PROGRAM P_Machine 

VAR	
	// MachineConfig
	stCurMachineConfig				: ST_MachineConfig;
	fOverride						: LREAL;
	bCheckPosBeforeRun				: BOOL;
	
	/// Sequences	
	seqOpMode						: FB_Sequence;
	
	bMaintMat						: BOOL;
	bMaintTool						: BOOL;
	stPunchJob						: ST_PunchJob;
		
	/// Components	
	fbComponents					: FB_CompositionBase;

	// PunchParameters
	bMatLoaded						: BOOL;
	bContinuous						: BOOL;
	nCurRun							: UINT;
	nCurPunch						: UDINT;
	nCurMat							: UINT;	
	nCurMoveOverride				: REAL;
	
	fThresholdX						: LREAL;
	fThresholdY						: LREAL;
	
	stCoordinate					: ST_Coordinate;
	stNextCoordinate				: ST_Coordinate;
	nMaxPunches						: UDINT;
	
	fMaxDisplacementX				: LREAL;
	fMaxDisplacementY				: LREAL;
	
	bInitialized					: BOOL;
	eJobState						: E_JobState;
	
	rtSafety						: R_TRIG;
	
	bSafeDrive						: BOOL;
	
	
END_VAR

// Init
Init();

bSafeDrive := fbSafety.SafetyOk AND fbSafetyLock.SafetyOk;

rtSafety(CLK:= NOT fbSafety.SafetyOk);

// SAFETY
IF rtSafety.Q THEN
	bInitialized := FALSE;
	seqOpMode.Start(E_OperationMode.eOperationMode_Halt);
	fbEventLog.WriteInfo(E_Event.eEvent_none, 'NOT HALT');
	
	IF eJobState = E_JobState.eJobState_running THEN
		eJobState := E_JobState.eJobState_stopped;
	END_IF
	
END_IF

// Run Components
fbEventLog.Run();
fbComponents.Run();

// Run Sequencer
seqOpMode.Enable := TRUE;
seqOpMode.Base(TRUE,FALSE);
CASE seqOpMode.SequenceId OF	
	E_OperationMode.eOperationMode_Maintenance:		_Maintenance();
	E_OperationMode.eOperationMode_Start:			_Start();
	E_OperationMode.eOperationMode_Stop:			_Stop();
	E_OperationMode.eOperationMode_Reset:			_Reset();
	E_OperationMode.eOperationMode_Halt:			_Halt();
END_CASE

METHOD _Halt : BOOL
VAR_INPUT
END_VAR
seqOpMode.Name := 'Halt';

CASE seqOpMode.Step OF
	
0	 :	seqOpMode.StepDefinition('Move to Zero Position', T#0S);
		fbPunchEngine.Halt();
		fbMatAndToolHandling.Halt();
		seqOpMode.NextStepDelay(T#1S, 10);	
		
10	 :	//fbSafetyLock.Unlock();
		seqOpMode.Finish();
		
END_CASE
END_METHOD

METHOD _Maintenance : BOOL
VAR_INPUT
END_VAR
seqOpMode.Name := 'Maintenance';

CASE seqOpMode.Step OF
	

0	 :	seqOpMode.StepDefinition('Move PunchEngine to Maint Position', T#0S);	
		fbPunchEngine.MoveTDC();			
		fbPunchEngine.OutletBeltseq(FALSE, 0);
		seqOpMode.NextStep(10);
	
10	 :	IF fbPunchEngine.TDC THEN
			seqOpMode.NextStep(20);		
		END_IF
		
20	 :	seqOpMode.StepDefinition('Move XY to Maint Position', T#0S);	
		fbMatAndToolHandling.MaintPos(NOT bMaintMat, NOT bMaintTool);	
		seqOpMode.NextStep(30);			
	
30	 :	IF fbMatAndToolHandling.TargetReached THEN 	
			seqOpMode.Finish();		
			//fbSafetyLock.Unlock();
		END_IF

			
END_CASE
END_METHOD

METHOD _Reset : BOOL
VAR_INPUT
END_VAR
CASE seqOpMode.Step OF

	0:	seqOpMode.StepDefinition('reset, init reset WF', T#0S);
		
		fbSafetyLock.Lock();
		bInitialized := FALSE;
		fbComponents.ResetComponents(FALSE, FALSE, 0, 0);
		
		fbEventLog.Mute := TRUE;
		fbEventLog.Reset();	
		
		seqOpMode.NextStepDelay(T#200MS, 10);	// skip safety

	10:	seqOpMode.StepDefinition('Reset: wait for request', T#0S);
		fbSafety.Reset();
		seqOpMode.NextStep(20);
		
	20:	seqOpMode.StepDefinition('Reset safety', T#0S);
		seqOpMode.NextStepTransition(30, fbSafety.State = E_ComponentState.eComponentState_running);
	
	30:	seqOpMode.StepDefinition('Reset all components', T#0S);
		fbComponents.ResetComponents(FALSE, FALSE, eComponentType_none, eComponentType_Safety);
		seqOpMode.NextStep(40);
		
	40:	seqOpMode.StepDefinition('wait for components ready...', T#0S);
		seqOpMode.NextStepTransitionDelay(fbComponents.CompostitionState = E_ComponentState.eComponentState_running, T#5S,  50);
		
	50:	seqOpMode.StepDefinition('Move to Zero Position', T#0S);
		fbPunchEngine.MoveTDC();
		fbPunchEngine.OutletBeltseq(FALSE, 0);
		seqOpMode.NextStep(60);	
		
	60:	IF fbPunchEngine.TDC THEN
			seqOpMode.NextStep(70);	
		END_IF
			
	70:	seqOpMode.StepDefinition('Finish', T#0S);
		fbEventLog.Mute := FALSE;
		fbEventLog.Reset();
		bInitialized := TRUE;
		seqOpMode.Finish();
		
END_CASE
END_METHOD

METHOD _Start : BOOL
VAR
	fTime				: LREAL;
	stTmpPosition		: ST_Coordinate;
END_VAR
seqOpMode.Name := 'Start';

CASE seqOpMode.Step OF
	
/// MAT LOOP

0	 :	seqOpMode.StepDefinition('Check Mat', T#0S);
		
		fbSafetyLock.Lock();
		IF NOT bInitialized THEN			// AUTO INIT
			seqOpMode.NextSequenceId := eOperationMode_Start;
			seqOpMode.Start(E_operationMode.eOperationMode_Reset);
			RETURN;
		END_IF
		
		IF NOT fbMatAndToolHandling.Ready OR NOT fbPunchEngine.Ready THEN
			RETURN;
		END_IF

		IF nCurMat > MATS_COUNT THEN
			fbPunchEngine.MoveTDC();
			fbMatAndToolHandling.MoveRelX(stCurMachineConfig.fMoveOutside ,stCurMachineConfig.fVelocityX, stCurMachineConfig.fAccelerationX);
			fbEventLog.WriteInfo(E_Event.eEvent_none, 'no further Mat Found');
			seqOpMode.NextStep(5);		
			RETURN;
		END_IF		

		IF stPunchJob.abMultipleMats[nCurMat] THEN
			fbMatAndToolHandling.SetupMat(fbMat.Mat.astMatOrigins[nCurMat]);	
			fbPunchEngine.MoveTDC();
			seqOpMode.NextStep(10);
		ELSE	
			nCurMat:= nCurMat + 1;
		END_IF	
		
5	 :	seqOpMode.StepDefinition('Finish Job', T#0S);
		IF fbMatAndToolHandling.TargetReached AND fbPunchEngine.TDC THEN
			fbPunchEngine.OutletBeltOnce();		
			eJobState := E_JobState.eJobState_finished;
			Halt();
		END_IF
		
10	 :	seqOpMode.StepDefinition('Move PunchEngine to Zero Position', T#0S);
		IF fbPunchEngine.TDC THEN
			seqOpMode.NextStep(20);		
		END_IF

/// RUN LOOP		
		
20	 :	seqOpMode.StepDefinition('Check Run if active', T#0S);		
		IF nCurRun > MATRUNS_COUNT THEN
			fbEventLog.WriteInfo(E_Event.eEvent_none, 'no further Run Found');
			nCurMat:= nCurMat + 1;
			nCurRun := 0;		
			seqOpMode.NextStep(0);
			RETURN;
		END_IF

		CASE stPunchJob.astRunTodo[nCurRun] OF			
			E_RunTodo.Punch_Tool_1:	
				fbMatAndToolHandling.SetupToolholder(1,fbMat.Mat.astRuns[nCurRun].stToolHolder.fX_Offset, fbMat.Mat.astRuns[nCurRun].stToolHolder.fY_Offset);
				fbMatAndToolHandling.ChangeTool(1);
				seqOpMode.NextStep(30);	
			
			E_RunTodo.Punch_Tool_2:	
				fbMatAndToolHandling.SetupToolholder(2,fbMat.Mat.astRuns[nCurRun].stToolHolder.fX_Offset, fbMat.Mat.astRuns[nCurRun].stToolHolder.fY_Offset);
				fbMatAndToolHandling.ChangeTool(2);
				seqOpMode.NextStep(30);		
				
			ELSE
				nCurRun := nCurRun + 1;			
		END_CASE

30	 :	seqOpMode.StepDefinition('Changing Tool', T#0S);
		IF fbMatAndToolHandling.ToolChanged THEN
			seqOpMode.NextStep(40);
		END_IF
		
40	 :	seqOpMode.StepDefinition('Prepare Data of current Run', T#0S);
		nMaxPunches := fbMat.Count_HolesOfRun(nCurRun);			
		fMaxDisplacementX	:= 0;
		fMaxDisplacementY	:= 0;
		
		
		// get Coordiantes of MatRun
		IF fbMat.SortRun(nCurRun) <> E_OperationResult.eOperationResult_Ok THEN		
			fbEventLog.WriteWarning(E_Event.eEvent_none, 'Error while sorting Coordinate-Array', FALSE);
			seqOpMode.Finish();
			RETURN;
		END_IF
				
		IF fbMat.ResortCoordinates(E_CoordinatesSortState.eCoordinatesSortState_resorted_v1) <> E_OperationResult.eOperationResult_Ok THEN
			fbEventLog.WriteWarning(E_Event.eEvent_none, 'Error while resorting Coordinate-Array', FALSE);
			seqOpMode.Finish();
			RETURN;
		END_IF
				

		// Set/Calc Override, Velocity, Acceleratopn of Punch	
		nCurMoveOverride := SEL(fbMat.Mat.astRuns[nCurRun].fMoveOverride = 0, INT_TO_REAL(fbMat.Mat.astRuns[nCurRun].fMoveOverride), 100)/100;
		
		fThresholdX:= SEL(fbMat.Mat.astRuns[nCurRun].fThresholdX = -1, fbMat.Mat.astRuns[nCurRun].fThresholdX, fbMat.MaxDistanceX);
		fThresholdY:= SEL(fbMat.Mat.astRuns[nCurRun].fThresholdY = -1, fbMat.Mat.astRuns[nCurRun].fThresholdY, fbMat.MaxDistanceY);
		fTime := fbMatAndToolHandling.GetMovementTime(  fThresholdX, 
													    fThresholdY,
														stCurMachineConfig.fVelocityX,
														stCurMachineConfig.fAccelerationX*nCurMoveOverride, 
														stCurMachineConfig.fVelocityY,
														stCurMachineConfig.fAccelerationY);	
		fbPunchEngine.SetupPunch(fbMat.Mat.fHeight, stCurMachineConfig.fSaftyDistanceToMat, stCurMachineConfig.fVelocityPunch, stCurMachineConfig.fAccelerationPunch, fTime);
		Override := SEL(fbMat.Mat.astRuns[nCurRun].fPunchOverride = 0, fbMat.Mat.astRuns[nCurRun].fPunchOverride, 100);
		
		// Calculate Coordinates		
		IF fbMat.GetCoordinate(nCurRun, nCurPunch, ADR(stCoordinate)) = E_OperationResult.eOperationResult_NOk THEN
			fbEventLog.WriteWarning(E_Event.eEvent_none, 'Error in getting Coordinate', FALSE);
			seqOpMode.Finish();
			RETURN;
		END_IF	
		
		stCoordinate.fX := stCoordinate.fX + stCurMachineConfig.stMatOrigin.fX;	
		stCoordinate.fY := stCoordinate.fY + stCurMachineConfig.stMatOrigin.fY;		
		
		
		// Move to Coordinate
		stTmpPosition := stCoordinate;
		stTmpPosition.fX := stTmpPosition.fX - stCurMachineConfig.fPassDistance;
		fbMatAndToolHandling.MoveAbs(	stTmpPosition, 
										stCurMachineConfig.fVelocityX, 
										stCurMachineConfig.fAccelerationX, 
										stCurMachineConfig.fVelocityY, 
										stCurMachineConfig.fAccelerationY);	

			
		seqOpMode.NextStep(45);		
		
45	 : 	seqOpMode.StepDefinition('Start from the same Direction', T#0S);
		IF fbMatAndToolHandling.TargetReached THEN
			fbMatAndToolHandling.MoveAbs(	stCoordinate, 
											stCurMachineConfig.fVelocityX, 
											stCurMachineConfig.fAccelerationX*nCurMoveOverride, 
											stCurMachineConfig.fVelocityY, 
											stCurMachineConfig.fAccelerationY);			
			seqOpMode.NextStep(50);		
		END_IF	
			
50	 : 	seqOpMode.StepDefinition('Move to First Position Before Loop', T#0S);
		IF fbMatAndToolHandling.TargetReached AND NOT bCheckPosBeforeRun THEN	
			seqOpMode.NextStep(60);		
		END_IF		
		
		IF seqOpMode.NextSequence THEN
			seqOpMode.Finish();
			RETURN;
		END_IF		
		
// PUNCHING LOOP
	
60	 :	seqOpMode.StepDefinition('Preparing', T#0S);
		IF fbMat.GetCoordinate(nCurRun, nCurPunch, ADR(stCoordinate)) = E_OperationResult.eOperationResult_NOk THEN
			fbEventLog.WriteWarning(E_Event.eEvent_none, 'Error in getting Coordinate', FALSE);
			seqOpMode.Finish();
			RETURN;
		END_IF	
		
		// outletbelt	
		IF fbMat.Mat.astRuns[nCurRun].bOutletbelt THEN
			fbPunchEngine.OutletBeltSeq(TRUE, fbMat.Mat.astRuns[nCurRun].nOutletbeltIntervall);
		END_IF
		
		// get next Coordinate	
		fbMat.GetCoordinate(nCurRun, nCurPunch+1, ADR(stNextCoordinate));
			
		IF seqOpMode.NextSequence THEN
			bContinuous := FALSE;
		ELSIF nCurPunch + 1 >= nMaxPunches THEN
			bContinuous := FALSE;
		ELSIF ABS(stNextCoordinate.fX - stCoordinate.fX) <= (fThresholdX + 0.1)				/// Nummerischer Fehler beim Berechnen des Treshholds wird mit 0.1 ausgeglichen 
		  AND ABS(stNextCoordinate.fY - stCoordinate.fY) <= (fThresholdY + 0.1) THEN
			bContinuous := TRUE;
		ELSE
			bContinuous := FALSE;
		END_IF
		
		// Calculate Asolute Coordinates
		stCoordinate.fX := stCoordinate.fX + stCurMachineConfig.stMatOrigin.fX;
		stCoordinate.fY := stCoordinate.fY + stCurMachineConfig.stMatOrigin.fY;		
		
		// Move to Coordinate
		fbMatAndToolHandling.MoveAbs(	stCoordinate, 
										stCurMachineConfig.fVelocityX, 
										stCurMachineConfig.fAccelerationX*nCurMoveOverride, 
										stCurMachineConfig.fVelocityY, 
										stCurMachineConfig.fAccelerationY);		
										
		IF fbPunchEngine.Punching THEN
			fbPunchEngine.Punch(bContinuous);
			seqOpMode.NextStep(80);	
		ELSE
			seqOpMode.NextStep(70);			
		END_IF	
		
70	 :	seqOpMode.StepDefinition('Moving', T#0S);
		// Anforderung auf Operationsmoduswechsel
		IF seqOpMode.NextSequence THEN
			seqOpMode.Finish();
			RETURN;
		END_IF		


		IF fbMatAndToolHandling.TargetReached THEN	
			fbPunchEngine.Punch(bContinuous);
			seqOpMode.NextStep(80);		
		END_IF		
		
80	 :	seqOpMode.StepDefinition('Punching', T#0S);

		// Wenn nicht durchgehend gestanzt wird warten bis der Stanzprozess abgeschlossen ist
		IF NOT bContinuous AND fbPunchEngine.Punching THEN
			RETURN;
		END_IF
	
		// Überprüfe den Unterschied zwischen IST/SOLL Position -> FEHLER bei zu hohem Unterschied
		IF fbPunchEngine.PunchDone THEN		
			stTmpPosition := fbMatAndToolHandling.Position;
			fMaxDisplacementX := MAX(fMaxDisplacementX, ABS(stCoordinate.fX - stTmpPosition.fX));
			fMaxDisplacementY := MAX(fMaxDisplacementY, ABS(stCoordinate.fY - stTmpPosition.fY));	
			nCurPunch := nCurPunch + 1;
			seqOpMode.NextStep(60);	
		END_IF
		
		// Keine weitere Stanzung in diesem Durchgang 
		IF nCurPunch >= nMaxPunches THEN
			fbEventLog.WriteInfo(E_Event.eEvent_none, 'Run Finished');
			fbPunchEngine.OutletBeltSeq(FALSE, 0);
			nCurPunch := 0;
			nCurRun := nCurRun + 1;
			seqOpMode.NextStep(20);	
			RETURN;
		END_IF	
		

END_CASE
END_METHOD

METHOD _Stop : BOOL
VAR_INPUT
END_VAR
seqOpMode.Name := 'Stop';

CASE seqOpMode.Step OF
	
0	 :	seqOpMode.StepDefinition('Move Punch to Zero Position', T#0S);
		fbPunchEngine.MoveTDC();
		fbPunchEngine.OutletBeltOnce();
		seqOpMode.NextStep(10);	
		
10	 :	seqOpMode.StepDefinition('Move Punch to Zero Position', T#0S);	
		IF fbPunchEngine.TDC THEN
			seqOpMode.NextStep(20);	
		END_IF
	
20	 :	seqOpMode.StepDefinition('Move Y-Axis to Zero Position', T#0S);		
		fbMatAndToolHandling.MoveAbsY(10, stCurMachineConfig.fVelocityX, stCurMachineConfig.fAccelerationX); //TODO: not hardcoded Position
		seqOpMode.NextStep(30);	

30	 :  IF fbMatAndToolHandling.TargetReached THEN
			fbPunchEngine.OutletBeltOnce();	
			seqOpMode.NextStepDelay(T#1S, 40);	
		END_IF	
		
40	 :	seqOpMode.StepDefinition('Stop finished', T#0S);	
		//fbSafetyLock.Unlock();
		seqOpMode.Finish();
		
	
END_CASE
END_METHOD

PROPERTY CheckPosBeforeRun : BOOL
GET
CheckPosBeforeRun := bCheckPosBeforeRun;
END_GET
SET
bCheckPosBeforeRun := CheckPosBeforeRun;
END_SET
END_PROPERTY

METHOD ClearJob : BOOL
VAR_INPUT
END_VAR
nCurRun := 0;
nCurPunch := 0;
nCurMat := 0;
MEMSET(ADR(stPunchJob), 0, SIZEOF(stPunchJob));

eJobState := E_JobState.eJobState_none;
END_METHOD

PROPERTY CountAllHolesOfJob : UDINT
GET
VAR
	ni						: UINT;
	nMats					: UINT;
	nPunchCount				: UDINT;
END_VAR
IF NOT bMatLoaded THEN
	RETURN;
END_IF

nMats := 0;
FOR ni := 0 TO MATS_COUNT DO
	IF 	stPunchJob.abMultipleMats[ni] THEN
		nMats := nMats + 1;
	END_IF
END_FOR

IF nMats = 0 THEN
	RETURN;
END_IF

nPunchCount := 0;
FOR ni := 0 TO MATRUNS_COUNT DO
	IF stPunchJob.astRunTodo[ni] = 0 THEN
		CONTINUE;
	END_IF
	nPunchCount := nPunchCount + fbMat.Count_HolesOfRun(ni);
END_FOR

CountAllHolesOfJob := nPunchCount * nMats;
END_GET
END_PROPERTY

PROPERTY CountRemainHolesOfJob : UDINT
GET
VAR
	ni						: UINT;
	nMats					: UINT;
	nPunchCount				: UDINT;
END_VAR
IF NOT bMatLoaded THEN
	RETURN;
END_IF

nMats := 0;
FOR ni := nCurMat TO MATS_COUNT DO
	IF 	stPunchJob.abMultipleMats[ni] THEN
		nMats := nMats + 1;
	END_IF
END_FOR

IF nMats = 0 THEN
	RETURN;
END_IF

nPunchCount := 0;
FOR ni := nCurRun TO MATRUNS_COUNT DO
	IF stPunchJob.astRunTodo[ni] = 0 THEN
		CONTINUE;
	END_IF
	nPunchCount := nPunchCount + fbMat.Count_HolesOfRun(ni);
END_FOR

CountRemainHolesOfJob := nPunchCount * nMats - nCurPunch;
END_GET
END_PROPERTY

PROPERTY CurMat : UINT
GET
CurMat := nCurMat;
END_GET
END_PROPERTY

PROPERTY CurPunch : UDINT
GET
CurPunch := nCurPunch;
END_GET
END_PROPERTY

PROPERTY CurRun : UINT
GET
CurRun := nCurRun;
END_GET
END_PROPERTY

METHOD Halt : E_OperationResult
VAR_INPUT
END_VAR
Halt := E_OperationResult.eOperationResult_NOk;

//ClearJob();
seqOpMode.Start(E_OperationMode.eOperationMode_Halt);

Halt := E_OperationResult.eOperationResult_Ok;
END_METHOD

METHOD Init : BOOL
VAR
	stLogConfig						: ST_LoggingConfig;
	stPlcAppSystemInfo				: PlcAppSystemInfo;
END_VAR

VAR_STAT
	OnlineChangesMirror				: UDINT;		
	FirstRun						: BOOL := TRUE;
END_VAR
//Init on OnlineChange
stPlcAppSystemInfo := Statics.stPlcSystemInfo.stPlcAppSystemInfo;
IF OnlineChangesMirror <> stPlcAppSystemInfo.OnlineChangeCnt OR FirstRun THEN
	OnlineChangesMirror := stPlcAppSystemInfo.OnlineChangeCnt;
	FirstRun := FALSE;
	
	InitComponents();
	InitConfig();

END_IF
END_METHOD

METHOD InitComponents : BOOL
VAR
	stLogConfig						: ST_LoggingConfig;
END_VAR
// Eventlog
stLogConfig.eLoggingProvider := E_LoggingProvider.eLoggingProviderEventLog;	
stLogConfig.sLogName := 'Punch.log';	
stLogConfig.sLogPath := 'C:\Log\Punch';									
stLogConfig.eLogLevel := E_LogLevel.eLogLevelInformation; 				
fbEventLog.Config := stLogConfig;
fbEventLog.Reset();

fbComponents.LoadComponents();	
fbComponents.Active := TRUE;
fbComponents.Name := 'Collection of all Components';
fbComponents.SetEventLogReference(fbEventLog);	

/// Supervison
fbComponents.RegisterComponent(1, fbSupervision);
fbSupervision.Active := TRUE;
fbSupervision.Name := 'Supervision';
fbSupervision.MachineArea := .eMachineArea_common;

/// Ethercat-Bus
fbComponents.RegisterComponent(2, fbEtherCATBus);
fbEtherCATBus.Active := TRUE;
fbEtherCATBus.Name := 'EtherCAT Bus';
fbEtherCATBus.MachineArea := E_MachineArea.eMachineArea_common;
fbEtherCATBus.SetReferences(COMP.stEtherCATState);

/// Safety
fbComponents.RegisterComponent(3, fbSafety);
fbSafety.Active := TRUE;
fbSafety.Name := 'Safety';
fbSafety.MachineArea := E_MachineArea.eMachineArea_common;
fbSafety.SetReferences(COMP.stSafetyIO);

/// Mat
fbComponents.RegisterComponent(5, fbMat);
fbMat.Active := TRUE;
fbMat.Name := 'Mat Definition';
fbMat.MachineArea := E_MachineArea.eMachineArea_common;

/// Mat and Tool Handling
fbComponents.RegisterComponent(6, fbMatAndToolHandling);
fbMatAndToolHandling.Active := TRUE;
fbMatAndToolHandling.Name := 'Mat and Tool Handling';
fbMatAndToolHandling.MachineArea := E_MachineArea.eMachineArea_common;
fbMatAndToolHandling.Setup(E_Axis.eAxis_X, E_Axis.eAxis_Y, E_Cylinder.eCylinder_Toolselector);
//fbMatAndToolHandling.Override := 100;
fbMatAndToolHandling.SetupToolDistance(0, 278.7);
fbMatAndToolHandling.SetupEnable(bSafeDrive);

/// Punch Engine
fbComponents.RegisterComponent(4, fbPunchEngine);
fbPunchEngine.Active := TRUE;
fbPunchEngine.Name := 'Punch Engine';
fbPunchEngine.MachineArea := E_MachineArea.eMachineArea_common;
fbPunchEngine.Setup(E_Axis.eAxis_Punch, E_DigitalOutput.eDigitalOutput_OutletBelt);
//fbPunchEngine.Override := 100;
fbPunchEngine.SetupCrank(420, 20);
fbPunchEngine.SetupEnable(bSafeDrive);


/// Safety Lock
fbComponents.RegisterComponent(4, fbSafetyLock);
fbSafetyLock.Active := TRUE;
fbSafetyLock.Name := 'Punch Engine';
fbSafetyLock.MachineArea := E_MachineArea.eMachineArea_common;
fbSafetyLock.SetReferences(COMP.stSafetyLockIO);

Override := 10;

/// Add Log
fbEventLog.Logger.AddLog('System startup, configuration loaded.', sName, E_LogLevel.eLogLevelInformation);
END_METHOD

METHOD InitConfig : BOOL
VAR
	stConfig				: ST_MachineConfig;
END_VAR
stConfig.stMatOrigin.fX := -20.5;
stConfig.stMatOrigin.fY := 343.5;

stConfig.fAccelerationX := 11000;//5500/2;
stConfig.fAccelerationY := 11000;//11000/2;
stConfig.fAccelerationPunch := 11000;

stConfig.fVelocityX := 660;
stConfig.fVelocityY := 660;
stConfig.fVelocityPunch := 900;

stConfig.fSaftyDistanceToMat := 0;

stConfig.stMaintPosition.fX := 10;
stConfig.stMaintPosition.fY := 10;
stConfig.stMaintPositionAlt.fX := 4050;
stConfig.stMaintPositionAlt.fY := 10;

stConfig.fMoveOutside := 440;
stConfig.fPassDistance := 2;

stConfig.nPunchTorqueLimit := 100;
stConfig.nPunchTorqueLimitNeg := 20;
stConfig.nPunchTorqueLimitPos := 100;

stConfig.nXTorqueLimit := 50;
stConfig.nYTorqueLimit := 100;

LoadConfig(stConfig);
END_METHOD

PROPERTY JobState : E_Jobstate
GET
VAR
	ni						: UINT;	
	bCheck					: BOOL;
END_VAR
JobState := eJobState;

//JobState := E_JobState.eJobState_error;
//
//// check if there ist at least one Mat enabled
//bCheck := FALSE;
//FOR ni := 0 TO MATS_COUNT DO
//	IF 	stPunchJob.abMultipleMats[ni] THEN
//		bCheck := TRUE;
//		EXIT;
//	END_IF
//	CONTINUE;
//END_FOR
//IF NOT bCheck THEN
//	RETURN;
//END_IF
//
//// check if there ist at least one Run enabled
//bCheck := FALSE;
//FOR ni := 0 TO MATRUNS_COUNT DO	
//	IF stPunchJob.astRunTodo[ni] <> 0 THEN
//		bCheck := TRUE;
//		EXIT;
//	END_IF
//	CONTINUE;
//END_FOR
//IF NOT bCheck THEN
//	RETURN;
//END_IF
//
//// check differences between Todolist and mat
//FOR ni := 0 TO MATRUNS_COUNT DO
//	IF stPunchJob.astRunTodo[ni] <> 0 AND NOT fbMat.Mat.astRuns[ni].bActive THEN
//		RETURN;
//	END_IF
//END_FOR
//
//
//JobState := E_JobState.eJobState_ready;
//
//IF seqOpMode.SequenceId = eOperationMode_Start AND seqOpMode.State = eSequenceState_running THEN
//	JobState := E_JobState.eJobState_running;
//END_IF
//
//IF nCurRun + nCurPunch + nCurMat = 0 THEN
//	JobState := E_JobState.eJobState_stopped;
//END_IF
END_GET
END_PROPERTY

METHOD LoadConfig : E_OperationResult
VAR_INPUT
	stConfig				: ST_MachineConfig;
END_VAR
LoadConfig := E_OperationResult.eOperationResult_NOk;

stCurMachineConfig := stConfig;

fbPunchEngine.TorqueLimit := stCurMachineConfig.nPunchTorqueLimit;
fbPunchEngine.TorqueLimitNeg := stCurMachineConfig.nPunchTorqueLimitNeg;
fbPunchEngine.TorqueLimitPos := stCurMachineConfig.nPunchTorqueLimitPos;

fbMatAndToolHandling.TorqueLimitX := stCurMachineConfig.nXTorqueLimit;
fbMatAndToolHandling.TorqueLimitY := stCurMachineConfig.nYTorqueLimit;

LoadConfig := E_OperationResult.eOperationResult_Ok;
END_METHOD

METHOD LoadJob : E_OperationResult
VAR_INPUT
	PunchJob				: ST_PunchJob;
END_VAR

VAR
	ni						: UINT;	
	bCheck					: BOOL;
END_VAR
LoadJob := E_OperationResult .eOperationResult_NOk;

// CHECK IF SAME
//IF MEMCMP(ADR(PunchJob), ADR(stPunchJob), SIZEOF(ST_PunchJob)) = 0 THEN
//	LoadJob := E_OperationResult .eOperationResult_Ok;
//	RETURN;
//END_IF

IF eJobState = E_JobState.eJobState_running OR eJobState = E_JobState.eJobState_stopped THEN
	RETURN;
END_IF

// check if Mat is loaded
IF NOT bMatLoaded THEN
	RETURN;
END_IF



// check if there ist at least one Mat enabled
bCheck := FALSE;
FOR ni := 0 TO MATS_COUNT DO
	IF 	PunchJob.abMultipleMats[ni] THEN
		bCheck := TRUE;
		EXIT;
	END_IF
	CONTINUE;
END_FOR
IF NOT bCheck THEN
	RETURN;
END_IF

// check if there ist at least one Run enabled
bCheck := FALSE;
FOR ni := 0 TO MATRUNS_COUNT DO	
	IF PunchJob.astRunTodo[ni] <> 0 THEN
		bCheck := TRUE;
		EXIT;
	END_IF
	CONTINUE;
END_FOR
IF NOT bCheck THEN
	RETURN;
END_IF

// check differences between Todolist and mat
FOR ni := 0 TO MATRUNS_COUNT DO
	IF PunchJob.astRunTodo[ni] <> 0 AND NOT fbMat.Mat.astRuns[ni].bActive THEN
		RETURN;
	END_IF
END_FOR

stPunchJob := PunchJob;	
eJobState := E_JobState.eJobState_ready;

LoadJob := E_OperationResult .eOperationResult_Ok;
END_METHOD

METHOD LoadMat : E_OperationResult
VAR_IN_OUT
	Mat						: ST_Mat;
END_VAR
VAR
	bMatOkay				: BOOL;
	ni						: UINT;
END_VAR
LoadMat := E_OperationResult.eOperationResult_NOk;

bMatLoaded := FALSE;
bMatOkay := FALSE;

IF Mat.fLenght = 0 OR Mat.fWidth = 0 THEN
	RETURN;
END_IF

FOR ni := 0 TO MATRUNS_COUNT DO
	
	// check if there is at lest one active Run
	IF  Mat.astRuns[ni].bActive THEN
		bMatOkay := TRUE;
		EXIT;
	END_IF
	
END_FOR

IF NOT bMatOkay THEN
	RETURN;
END_IF

fbMat.LoadMat(Mat);

bMatLoaded := TRUE;
LoadMat := E_OperationResult.eOperationResult_Ok;
END_METHOD

PROPERTY MachineConfig : ST_MachineConfig
GET
MachineConfig := stCurMachineConfig;
END_GET
SET
stCurMachineConfig := MachineConfig;
END_SET
END_PROPERTY

METHOD Maint : E_OperationResult
VAR_INPUT
	Mat				: BOOL;
	Tool			: BOOL;
	Alt				: BOOL;
END_VAR
Maint := E_OperationResult.eOperationResult_NOk;

IF eJobState = E_JobState.eJobState_running THEN
	eJobState := E_JobState.eJobState_stopped;
END_IF
seqOpMode.NextSequenceId := E_OperationMode.eOperationMode_Maintenance;

// load actual Maintposition
IF Alt THEN
	fbMatAndToolHandling.SetupMaintPos(stCurMachineConfig.stMaintPositionAlt);
ELSE
	fbMatAndToolHandling.SetupMaintPos(stCurMachineConfig.stMaintPosition);
END_IF
bMaintMat := Mat;
bMaintTool := Tool;

Maint := E_OperationResult.eOperationResult_Ok;
END_METHOD

PROPERTY MatLoaded : BOOL
GET
MatLoaded := bMatLoaded;
END_GET
END_PROPERTY

PROPERTY MatOriginX : REAL
GET
MatOriginX := stCurMachineConfig.stMatOrigin.fX;
END_GET
SET
stCurMachineConfig.stMatOrigin.fX := MatOriginX;
END_SET
END_PROPERTY

PROPERTY MatOriginY : REAL
GET
MatOriginY := stCurMachineConfig.stMatOrigin.fY;
END_GET
SET
stCurMachineConfig.stMatOrigin.fY := MatOriginY;
END_SET
END_PROPERTY

PROPERTY MaxPunch : UDINT
GET
MaxPunch := nMaxPunches;
END_GET
END_PROPERTY

PROPERTY Override : Lreal
GET
Override := fOverride;
END_GET
SET
fOverride := Override;
fbPunchEngine.Override := Override;
END_SET
END_PROPERTY

PROPERTY Punching : BOOL
GET
Punching := seqOpMode.SequenceId = eOperationMode_Start AND seqOpMode.State = eSequenceState_running ;
END_GET
END_PROPERTY

PROPERTY RemainTimeOfJob : UDINT
GET
IF fbPunchEngine.Velocity = 0 OR fOverride = 0 THEN
	RETURN;
END_IF

IF NOT Punching THEN
	RETURN;
END_IF

RemainTimeOfJob := LREAL_TO_UDINT(CountRemainHolesOfJob/(fbPunchEngine.Velocity/360)/fOverride*100/60);
END_GET
END_PROPERTY

METHOD Reset : E_OperationResult
VAR_INPUT
END_VAR
Reset := E_OperationResult.eOperationResult_NOk;

IF eJobState = E_JobState.eJobState_running THEN
	eJobState := E_JobState.eJobState_stopped;
END_IF
seqOpMode.Start(e_Operationmode.eOperationMode_Reset);

Reset := E_OperationResult.eOperationResult_Ok;
END_METHOD

METHOD Resume : E_OperationResult
VAR_INPUT
END_VAR

VAR
	ni						: UINT;	
	bCheck					: BOOL;
END_VAR
Resume := E_OperationResult.eOperationResult_NOk;

IF eJobState <> E_JobState.eJobState_ready AND eJobState <> E_JobState.eJobState_stopped THEN
	RETURN;
END_IF;;

IF Override = 0 THEN
	RETURN;
END_IF

eJobState := E_JobState.eJobState_running;
seqOpMode.Start(e_Operationmode.eOperationMode_Start);
Resume := E_OperationResult.eOperationResult_Ok;
END_METHOD

PROPERTY ResumeAllowed : BOOL
GET
VAR
	ni						: UINT;	
	bCheck					: BOOL;
END_VAR
ResumeAllowed := TRUE;

IF Punching THEN
	ResumeAllowed := FALSE;
	RETURN;	
END_IF

IF nCurRun + nCurPunch + nCurMat = 0 THEN
	ResumeAllowed := FALSE;
	RETURN;	
END_IF

// check if Mat is loaded
IF NOT bMatLoaded THEN
	ResumeAllowed := FALSE;
	RETURN;
END_IF

// check if there ist at least one Mat enabled
bCheck := FALSE;
FOR ni := 0 TO MATS_COUNT DO
	IF 	stPunchJob.abMultipleMats[ni] THEN
		bCheck := TRUE;
		EXIT;
	END_IF
	CONTINUE;
END_FOR
IF NOT bCheck THEN
	ResumeAllowed := FALSE;
	RETURN;
END_IF

// check if there ist at least one Run enabled
bCheck := FALSE;
FOR ni := 0 TO MATRUNS_COUNT DO	
	IF stPunchJob.astRunTodo[ni] <> 0 THEN
		bCheck := TRUE;
		EXIT;
	END_IF
	CONTINUE;
END_FOR
IF NOT bCheck THEN
	ResumeAllowed := FALSE;
	RETURN;
END_IF

// check differences between Todolist and mat
FOR ni := 0 TO MATRUNS_COUNT DO
	IF stPunchJob.astRunTodo[ni] <> 0 AND NOT fbMat.Mat.astRuns[ni].bActive THEN
		ResumeAllowed := FALSE;
		RETURN;
	END_IF
END_FOR
END_GET
END_PROPERTY

METHOD Start : E_OperationResult
VAR_INPUT
	PunchJob				: ST_PunchJob;
END_VAR

VAR
	ni						: UINT;	
	bCheck					: BOOL;
END_VAR
Start := E_OperationResult.eOperationResult_NOk;

//IF fbSafetyLock.Opened THEN
//	RETURN;
//END_IF

ClearJob();
LoadJob(PunchJob);

IF Override = 0 THEN
	RETURN;
END_IF

eJobState := E_JobState.eJobState_running;
seqOpMode.Start(e_Operationmode.eOperationMode_Start);
Start := E_OperationResult.eOperationResult_Ok;
END_METHOD

METHOD Stop : E_OperationResult
VAR_INPUT
END_VAR
Stop := E_OperationResult.eOperationResult_NOk;

seqOpMode.NextSequenceId := E_OperationMode.eOperationMode_Stop;

IF eJobState = E_JobState.eJobState_running THEN
	eJobState := E_JobState.eJobState_stopped;
END_IF

Stop := E_OperationResult.eOperationResult_Ok;
END_METHOD

END_PROGRAM

(* stored: Version 1.1.0.1, ProductVersion 3.1.4022.12
   POU P_Machine: Id {0d8c50ec-918a-4b59-8662-1a71ca9d0388}, SpecialFunc None
   Folder Commands: Id {a3c3c167-6bae-43eb-9a17-ee7ed08c2459}
   Folder Init: Id {cd91c3b9-9472-40be-ac4b-a2f3e03535a6}
   Folder OpMode: Id {448a1300-4b08-45ae-8e7d-de4a05de0e2f}
   Folder Properties: Id {b605d9af-9bd3-4b7a-aaeb-943cf423fa8f}
   Folder Utilities: Id {043088c3-1de5-4927-9556-8f5875bcaa03}
   Method _Halt: Id {8d0cc817-fb11-4d04-b110-815d1ab018d5}
   Method _Maintenance: Id {abd94d62-471b-4022-9d8a-d646a4da430c}
   Method _Reset: Id {b7ea65e0-91e4-4978-951d-b3671362c880}
   Method _Start: Id {05d25d84-933c-490b-b706-1f4b0edc50bb}
   Method _Stop: Id {6183ad43-eef9-48a2-acec-0f977ca27297}
   Property CheckPosBeforeRun: Id {d1e8ce50-5236-41a0-a206-fca240d6a6d4}
   Get Get: Id {4a5e9e39-3857-4c8a-bd10-551b4a073418}
   Set Set: Id {9805bd54-545a-47ef-be74-dbe6db912555}
   Method ClearJob: Id {7dc5521b-7346-4d08-b6cd-22f877e745f2}
   Property CountAllHolesOfJob: Id {bcd541cf-b00f-47ca-be15-45867cffb802}
   Get Get: Id {fe27e395-0315-40c4-aa83-495f4ffcf7c4}
   Property CountRemainHolesOfJob: Id {e91f8ffb-8807-4020-80d9-c4c2746e5856}
   Get Get: Id {cc1207f5-9cfe-4f8c-840e-29195922b115}
   Property CurMat: Id {6ae330f2-62c1-417b-adea-4e858716c937}
   Get Get: Id {dab8f04e-a273-4cd3-a985-2c96e9aa8c81}
   Property CurPunch: Id {bf013849-d40f-4942-bc33-6f60ec39ae15}
   Get Get: Id {89ac6a9c-2a98-46ac-a230-3bbaba97c8e5}
   Property CurRun: Id {a552c20f-8cac-4544-9764-39fa183f1bc9}
   Get Get: Id {88b4c6bc-6865-4c6a-99cc-325992d3207e}
   Method Halt: Id {efddaa5b-9660-496c-a523-94c2986c5dee}
   Method Init: Id {5beb4bc6-6c7b-4b75-9b3b-07a0dc189c65}
   Method InitComponents: Id {073cd59f-ca6a-43ca-851c-8fedfb1ab58b}
   Method InitConfig: Id {d048fa18-b357-4d6d-ae0f-62e152306f2c}
   Property JobState: Id {5408bbc4-92b1-47a4-aaa7-e48a225272b6}
   Get Get: Id {bc8f731f-54d3-486c-bdc9-9fe6ed7fbd23}
   Method LoadConfig: Id {7cd22898-429a-4ef9-afac-ce883356c33b}
   Method LoadJob: Id {06b9ba9d-0e6f-4218-8f2f-11979597d5f0}
   Method LoadMat: Id {5368a477-ce06-442c-9236-a3910d39d411}
   Property MachineConfig: Id {e153bf89-3003-472c-96dd-edebbbdf5ae6}
   Get Get: Id {b36aac0a-98b0-4b86-b9b3-044c7700925f}
   Set Set: Id {5736b3e3-210a-4e49-b4fe-734cf8936bda}
   Method Maint: Id {1ce4f865-fa11-4f8e-80d7-e65b61200476}
   Property MatLoaded: Id {fbdd7173-1b91-4257-8f69-7d7585cff951}
   Get Get: Id {25acb863-6fa5-4556-9b09-9ee0563f94ce}
   Property MatOriginX: Id {efd07f67-86da-4559-a465-623dd826c051}
   Get Get: Id {9fd3da1e-55bd-4633-8325-269168ceaf91}
   Set Set: Id {3f45f4fd-f9b0-4230-b0ea-40dc0b8dc889}
   Property MatOriginY: Id {6204fe5a-1cb7-4f53-af23-27d4e83ddd53}
   Get Get: Id {29851ec2-f24c-4972-9d7f-a89d46673d9e}
   Set Set: Id {f559f516-85ee-4980-bb7c-c1bc0ce8ad1b}
   Property MaxPunch: Id {08fb3a28-1eda-4fba-bd61-541974b3f637}
   Get Get: Id {16ab66ef-5ee7-4618-9723-ea13b782e356}
   Property Override: Id {0add2759-3c97-4992-acf8-86154fb24036}
   Get Get: Id {d671ea66-b89c-423e-ab53-ac84404cb99d}
   Set Set: Id {d0a59103-7b1e-45c3-b193-7041761db0b2}
   Property Punching: Id {54d2b23c-9c84-4db4-9337-4ccdacb1887a}
   Get Get: Id {c6bfbe16-946b-48bb-a5c1-0544f877a627}
   Property RemainTimeOfJob: Id {0480b95d-adb6-410c-b530-e88fa29fd0f2}
   Get Get: Id {f55c467b-7c01-4467-9b54-a63dc31e99b9}
   Method Reset: Id {7f9e7617-df72-435e-9ceb-840bb7eb2c67}
   Method Resume: Id {cd1c608f-4754-4f3c-89f1-c84c9e7f7fd3}
   Property ResumeAllowed: Id {c0f1c1aa-2034-4954-8ea2-0fb8cb7fcbb9}
   Get Get: Id {44cbb1e5-922f-4d67-9c36-df72e5614181}
   Method Start: Id {14a28483-6bb7-478f-933c-4c5d4e0212ad}
   Method Stop: Id {491817b2-2fa0-4bbe-8b92-f0e2f2be4718} *)
